// TIA Portal V17 export
// export: Created 2023-02-14T02:49:53.1247675Z, ExportSetting WithDefaults, DisplayName Totally Integrated Automation Portal, DisplayVersion V17, DisplayName TIA Portal Openness, DisplayVersion V17, DisplayName TIA Portal Teamcenter Gateway, DisplayVersion V17, DisplayName TIA Portal Version Control Interface, DisplayVersion V17, DisplayName SINAMICS Startdrive Advanced, DisplayVersion V17, DisplayName SINAMICS Startdrive G130, G150, S120, S150, SINAMICS MV, S210, DisplayVersion V17, DisplayName SINAMICS Startdrive G110M, G120, G120C, G120D, G120P, G115D, DisplayVersion V17, DisplayName STEP 7 Professional, DisplayVersion V17, DisplayName STEP 7 Safety, DisplayVersion V17, DisplayName WinCC Professional, DisplayVersion V17
DATA_BLOCK "PUT_OSA_CIP"   // DB56
// stored: AutoNumber false, DBAccessibleFromOPCUA true, DBAccessibleFromWebserver true, InstanceOfName PUT_SFB, OfSystemLibElement PUT, OfSystemLibVersion 1.3
"PUT_SFB"
   // VAR_INPUT
   //    REQ : Bool;
   //    ID : Word;
   // END_VAR
   // VAR_OUTPUT
   //    DONE : Bool;
   //    ERROR : Bool;
   //    STATUS : Word;
   // END_VAR
   // VAR_IN_OUT
   //    ADDR_1 : Remote;
   //    ADDR_2 : Remote;
   //    ADDR_3 : Remote;
   //    ADDR_4 : Remote;
   //    SD_1 : Variant;
   //    SD_2 : Variant;
   //    SD_3 : Variant;
   //    SD_4 : Variant;
   // END_VAR
BEGIN
END_DATA_BLOCK
